(* IEC 61131-3 sources: beckhoffAutomationInterface/ST/Shark/Lib/Sequences/SubSequence, 11 files *)

(* ---- FB_BubblerPurgeCMSequence.st ---- *)
FUNCTION_BLOCK PUBLIC FB_BubblerPurgeCMSequence IMPLEMENTS I_TreeNode
VAR
    _seq : FB_SequenceNode;
    // Steps
    stepOpenBubbler  : FB_OpenValveNode;
    stepPurgeCM      : FB_MaterialPurgeCMSequence;
    stepCloseBubbler : FB_CloseValveNode;

    // Internal state
    _bInitialized    : BOOL := FALSE;
    _eSide           : E_GasSide;
    _nBubblerIndex   : DINT;
END_VAR

METHOD PUBLIC Init : BOOL
VAR_INPUT
    ipProvider      : I_HardwareProvider;
    eSide           : E_GasSide;
    nBubblerIndex   : DINT;
END_VAR
VAR
    ipCMBubblerValve : I_Valve;
END_VAR
    IF _bInitialized THEN
        IF _eSide = eSide AND _nBubblerIndex = nBubblerIndex THEN
            Init := TRUE;
            RETURN;
        END_IF
        _seq.ClearChildren();
        _bInitialized := FALSE;
    END_IF

    IF ipProvider = 0 THEN
        GVL_ErrorLogger.Logger.LogError('FB_BubblerPurgeCMSequence', E_ErrorId.ERR_GEN_NULL_POINTER, 'Provider is null');
        RETURN;
    END_IF
    _eSide := eSide;
    _nBubblerIndex := nBubblerIndex;

    // Resolve hardware
    ipCMBubblerValve := ipProvider.GetCMBubblerValve(eSide, nBubblerIndex);

    IF ipCMBubblerValve = 0 THEN
        GVL_ErrorLogger.Logger.LogError('FB_BubblerPurgeCMSequence', E_ErrorId.ERR_GEN_NULL_POINTER, 'Bubbler Valve not found');
        RETURN;
    END_IF

    stepOpenBubbler.Init(ipCMBubblerValve, sNodeName := 'OpenBubblerCMValve');
    _seq.AddChild(stepOpenBubbler);

    stepPurgeCM.Init(ipProvider, eSide);
    stepPurgeCM.NodeName := 'PurgeCMSequence';
    _seq.AddChild(stepPurgeCM);

    stepCloseBubbler.Init(ipCMBubblerValve, sNodeName := 'CloseBubblerCMValve');
    _seq.AddChild(stepCloseBubbler);

    _seq.sName := CONCAT('BubblerPurgeCM_Side', TO_STRING(eSide));
    _bInitialized := TRUE;
    Init := TRUE;
END_METHOD

METHOD PUBLIC SetParams
VAR_INPUT
    nPurgeCycles            : INT;
    rPurgeFlowRate          : LREAL;
    rPurgePressure          : LREAL;
    rEvacuationPressure     : LREAL;
    tPressurizationTimeout  : TIME;
    tEvacuationTimeout      : TIME;
END_VAR
    IF NOT _bInitialized THEN RETURN; END_IF

    stepPurgeCM.SetParams(
        nPurgeCycles           := nPurgeCycles,
        rPurgeFlowRate         := rPurgeFlowRate,
        rPurgePressure         := rPurgePressure,
        rEvacuationPressure    := rEvacuationPressure,
        tPressurizationTimeout := tPressurizationTimeout,
        tEvacuationTimeout     := tEvacuationTimeout
    );
END_METHOD

PROPERTY PUBLIC NodeName : STRING(50)
    GET
        NodeName := _seq.sName;
    END_GET
    SET
        _seq.sName := NodeName;
    END_SET
END_PROPERTY

METHOD Tick : ST_NodeResult
    IF NOT _bInitialized THEN
        Tick.eStatus := E_NodeStatus.FAILURE;
        Tick.bHasError := TRUE;
        Tick.stError.eErrorId := E_ErrorId.ERR_GEN_INITIALIZATION;
        Tick.stError.sSource := 'FB_BubblerPurgeCMSequence';
        Tick.stError.sMessage := 'Init must be called before Tick';
        Tick.sDescription := Tick.stError.sMessage;
        RETURN;
    END_IF

    Tick := _seq.Tick();
END_METHOD

{attribute 'estimated-stack-usage' := '500'}
METHOD Reset : BOOL
    Reset := _seq.Reset();
END_METHOD

{attribute 'estimated-stack-usage' := '500'}
METHOD Halt
    _seq.Halt();
END_METHOD

END_FUNCTION_BLOCK

(* ---- FB_BubblerPurgeHMSequence.st ---- *)
FUNCTION_BLOCK PUBLIC FB_BubblerPurgeHMSequence IMPLEMENTS I_TreeNode
VAR
    _seq : FB_SequenceNode;
    // Steps
    stepOpenBubbler  : FB_OpenValveNode;
    stepPurgeHM      : FB_MaterialPurgeHMSequence;
    stepCloseBubbler : FB_CloseValveNode;

    // Internal state
    _bInitialized    : BOOL := FALSE;
    _eSide           : E_GasSide;
    _nBubblerIndex   : DINT;
END_VAR

METHOD PUBLIC Init : BOOL
VAR_INPUT
    ipProvider      : I_HardwareProvider;
    eSide           : E_GasSide;
    nBubblerIndex   : DINT;
END_VAR
VAR
    ipHMBubblerValve : I_Valve;
END_VAR
    IF _bInitialized THEN
        IF _eSide = eSide AND _nBubblerIndex = nBubblerIndex THEN
            Init := TRUE;
            RETURN;
        END_IF
        _seq.ClearChildren();
        _bInitialized := FALSE;
    END_IF

    IF ipProvider = 0 THEN
        GVL_ErrorLogger.Logger.LogError('FB_BubblerPurgeHMSequence', E_ErrorId.ERR_GEN_NULL_POINTER, 'Provider is null');
        RETURN;
    END_IF
    _eSide := eSide;
    _nBubblerIndex := nBubblerIndex;

    // Resolve hardware
    ipHMBubblerValve := ipProvider.GetHMBubblerValve(eSide, nBubblerIndex);

    IF ipHMBubblerValve = 0 THEN
        GVL_ErrorLogger.Logger.LogError('FB_BubblerPurgeHMSequence', E_ErrorId.ERR_GEN_NULL_POINTER, 'Bubbler Valve not found');
        RETURN;
    END_IF

    stepOpenBubbler.Init(ipHMBubblerValve, sNodeName := 'OpenBubblerHMValve');
    _seq.AddChild(stepOpenBubbler);

    stepPurgeHM.Init(ipProvider, eSide);
    stepPurgeHM.NodeName := 'PurgeHMSequence';
    _seq.AddChild(stepPurgeHM);

    stepCloseBubbler.Init(ipHMBubblerValve, sNodeName := 'CloseBubblerHMValve');
    _seq.AddChild(stepCloseBubbler);

    _seq.sName := CONCAT('BubblerPurgeHM_Side', TO_STRING(eSide));
    _bInitialized := TRUE;
    Init := TRUE;
END_METHOD

METHOD PUBLIC SetParams
VAR_INPUT
    nPurgeCycles            : INT;
    rPurgeFlowRate          : LREAL;
    rPurgePressure          : LREAL;
    rFinalPressure          : LREAL;   // Operating pressure for final pressurization
    rEvacuationPressure     : LREAL;
    tPressurizationTimeout  : TIME;
    tEvacuationTimeout      : TIME;
END_VAR
    IF NOT _bInitialized THEN RETURN; END_IF

    stepPurgeHM.SetParams(
        nPurgeCycles           := nPurgeCycles,
        rPurgeFlowRate         := rPurgeFlowRate,
        rPurgePressure         := rPurgePressure,
        rFinalPressure         := rFinalPressure,
        rEvacuationPressure    := rEvacuationPressure,
        tPressurizationTimeout := tPressurizationTimeout,
        tEvacuationTimeout     := tEvacuationTimeout
    );
END_METHOD

PROPERTY PUBLIC NodeName : STRING(50)
    GET
        NodeName := _seq.sName;
    END_GET
    SET
        _seq.sName := NodeName;
    END_SET
END_PROPERTY

METHOD Tick : ST_NodeResult
    IF NOT _bInitialized THEN
        Tick.eStatus := E_NodeStatus.FAILURE;
        Tick.bHasError := TRUE;
        Tick.stError.eErrorId := E_ErrorId.ERR_GEN_INITIALIZATION;
        Tick.stError.sSource := 'FB_BubblerPurgeHMSequence';
        Tick.stError.sMessage := 'Init must be called before Tick';
        Tick.sDescription := Tick.stError.sMessage;
        RETURN;
    END_IF

    Tick := _seq.Tick();
END_METHOD

{attribute 'estimated-stack-usage' := '500'}
METHOD Reset : BOOL
    Reset := _seq.Reset();
END_METHOD

{attribute 'estimated-stack-usage' := '500'}
METHOD Halt
    _seq.Halt();
END_METHOD

END_FUNCTION_BLOCK

(* ---- FB_DepressurizeCMSequence.st ---- *)
FUNCTION_BLOCK PUBLIC FB_DepressurizeCMSequence IMPLEMENTS I_TreeNode
VAR
    _seq : FB_SequenceNode;
    // Steps
    stepOpenCMPurge      : FB_OpenValveNode;
    stepOpenCMVacuumIso  : FB_OpenValveNode;
    stepWaitCMVacuum     : FB_WaitForSensorNode;
    stepCloseCMVacuumIso : FB_CloseValveNode;
    stepCloseCMPurge     : FB_CloseValveNode;

    // Internal state
    _bInitialized        : BOOL := FALSE;
    _eSide               : E_GasSide;
END_VAR

VAR CONSTANT
    DEFAULT_VACUUM_THRESHOLD : LREAL := 1.0; // Bar - pressure below which vacuum is considered achieved
END_VAR

METHOD PUBLIC Init : BOOL
VAR_INPUT
    ipProvider     : I_HardwareProvider;
    eSide          : E_GasSide;
    tVacuumTimeout : TIME := T#30S;
END_VAR
VAR
    ipCMPurge     : I_Valve;
    ipCMVacuumIso : I_Valve;
    ipCMPressure  : I_Sensor;
END_VAR
    IF _bInitialized THEN
        IF _eSide = eSide THEN
            Init := TRUE;
            RETURN;
        END_IF
        _seq.ClearChildren();
        _bInitialized := FALSE;
    END_IF

    IF ipProvider = 0 THEN
        GVL_ErrorLogger.Logger.LogError('FB_DepressurizeCMSequence', E_ErrorId.ERR_GEN_NULL_POINTER, 'Provider is null');
        RETURN;
    END_IF
    _eSide := eSide;

    // Resolve hardware references
    ipCMPurge := ipProvider.GetCMPurgeValve(eSide);
    ipCMVacuumIso := ipProvider.GetCMVacuumIsoValve(eSide);
    ipCMPressure := ipProvider.GetCMPressureSensor(eSide);

    IF ipCMPurge = 0 OR ipCMVacuumIso = 0 OR ipCMPressure = 0 THEN
        GVL_ErrorLogger.Logger.LogError('FB_DepressurizeCMSequence', E_ErrorId.ERR_GEN_NULL_POINTER, 'Hardware reference is null');
        RETURN;
    END_IF

    // Evacuation: open path to exhaust, wait for vacuum, then close
    stepOpenCMPurge.Init(ipCMPurge, sNodeName := 'OpenCMPurge');
    _seq.AddChild(stepOpenCMPurge);

    stepOpenCMVacuumIso.Init(ipCMVacuumIso, sNodeName := 'OpenCMVacuumIso');
    _seq.AddChild(stepOpenCMVacuumIso);

    stepWaitCMVacuum.Init(
        ipSensor    := ipCMPressure,
        rTarget     := DEFAULT_VACUUM_THRESHOLD,
        eMode       := E_CompareMode.LESS_THAN,
        tTimeout    := tVacuumTimeout,
        sNodeName   := 'WaitCMVacuum'
    );
    _seq.AddChild(stepWaitCMVacuum);

    stepCloseCMVacuumIso.Init(ipCMVacuumIso, sNodeName := 'CloseCMVacuumIso');
    _seq.AddChild(stepCloseCMVacuumIso);

    stepCloseCMPurge.Init(ipCMPurge, sNodeName := 'CloseCMPurge');
    _seq.AddChild(stepCloseCMPurge);

    _seq.sName := CONCAT('DepressurizeCM_', TO_STRING(eSide));
    _bInitialized := TRUE;
    Init := TRUE;
END_METHOD

METHOD PUBLIC SetParams
VAR_INPUT
    rVacuumThreshold : LREAL;
    tTimeout         : TIME;
END_VAR
    IF NOT _bInitialized THEN RETURN; END_IF

    stepWaitCMVacuum.Target := rVacuumThreshold;
    stepWaitCMVacuum.Timeout := tTimeout;
END_METHOD

PROPERTY PUBLIC NodeName : STRING(50)
    GET
        NodeName := _seq.sName;
    END_GET
    SET
        _seq.sName := NodeName;
    END_SET
END_PROPERTY

METHOD Tick : ST_NodeResult
    IF NOT _bInitialized THEN
        Tick.eStatus := E_NodeStatus.FAILURE;
        Tick.bHasError := TRUE;
        Tick.stError.eErrorId := E_ErrorId.ERR_GEN_INITIALIZATION;
        Tick.stError.sSource := 'FB_DepressurizeCMSequence';
        Tick.stError.sMessage := 'Init must be called before Tick';
        Tick.sDescription := Tick.stError.sMessage;
        RETURN;
    END_IF

    Tick := _seq.Tick();
END_METHOD

{attribute 'estimated-stack-usage' := '500'}
METHOD Reset : BOOL
    Reset := _seq.Reset();
END_METHOD

{attribute 'estimated-stack-usage' := '500'}
METHOD Halt
    _seq.Halt();
END_METHOD

END_FUNCTION_BLOCK

(* ---- FB_DepressurizeHMSequence.st ---- *)
FUNCTION_BLOCK PUBLIC FB_DepressurizeHMSequence IMPLEMENTS I_TreeNode
VAR
    _seq : FB_SequenceNode;
    // Safety steps
    stepCloseNozzle      : FB_CloseValveNode;
    stepClosePCV         : FB_SetControllerNode;

    // Evacuation
    stepOpenHMVacuumIso  : FB_OpenValveNode;
    stepOpenHMPurge      : FB_OpenValveNode;
    stepWaitHMVacuum     : FB_WaitForSensorNode;
    stepCloseHMVacuumIso : FB_CloseValveNode;
    stepCloseHMPurge     : FB_CloseValveNode;

    // Internal state
    _bInitialized        : BOOL := FALSE;
    _eSide               : E_GasSide;
END_VAR

VAR CONSTANT
    DEFAULT_VACUUM_THRESHOLD : LREAL := 1.0; // Bar - pressure below which vacuum is considered achieved
END_VAR

METHOD PUBLIC Init : BOOL
VAR_INPUT
    ipProvider    : I_HardwareProvider;
    eSide         : E_GasSide;
    tVacuumTimeout : TIME := T#30S;
END_VAR
VAR
    ipNozzleIso   : I_Valve;
    ipPCV         : I_Controller;
    ipHMPurge     : I_Valve;
    ipHMVacuumIso : I_Valve;
    ipHMPressure  : I_Sensor;
END_VAR
    IF _bInitialized THEN
        IF _eSide = eSide THEN
            Init := TRUE;
            RETURN;
        END_IF
        _seq.ClearChildren();
        _bInitialized := FALSE;
    END_IF

    IF ipProvider = 0 THEN
        GVL_ErrorLogger.Logger.LogError('FB_DepressurizeHMSequence', E_ErrorId.ERR_GEN_NULL_POINTER, 'Provider is null');
        RETURN;
    END_IF
    _eSide := eSide;

    // Resolve hardware references
    ipNozzleIso := ipProvider.GetNozzleIsoValve(eSide);
    ipPCV := ipProvider.GetPressureController(eSide);
    ipHMPurge := ipProvider.GetHMPurgeValve(eSide);
    ipHMVacuumIso := ipProvider.GetHMVacuumIsoValve(eSide);
    ipHMPressure := ipProvider.GetHMPressureSensor(eSide);

    IF ipNozzleIso = 0 OR ipPCV = 0 OR ipHMPurge = 0 OR ipHMVacuumIso = 0 OR ipHMPressure = 0 THEN
        GVL_ErrorLogger.Logger.LogError('FB_DepressurizeHMSequence', E_ErrorId.ERR_GEN_NULL_POINTER, 'Hardware reference is null');
        RETURN;
    END_IF

    // Safety: isolate nozzle and close PCV
    stepCloseNozzle.Init(ipNozzleIso, sNodeName := 'CloseNozzle');
    _seq.AddChild(stepCloseNozzle);

    stepClosePCV.Init(ipController := ipPCV, rSetpoint := GVL_SequenceConstants.PCV_CLOSED_SETPOINT, sNodeName := 'ClosePCV');
    _seq.AddChild(stepClosePCV);

    // Evacuation: open path to exhaust, wait for vacuum, then close
    stepOpenHMVacuumIso.Init(ipHMVacuumIso, sNodeName := 'OpenHMVacuumIso');
    _seq.AddChild(stepOpenHMVacuumIso);

    stepOpenHMPurge.Init(ipHMPurge, sNodeName := 'OpenHMPurge');
    _seq.AddChild(stepOpenHMPurge);

    stepWaitHMVacuum.Init(
        ipSensor    := ipHMPressure,
        rTarget     := DEFAULT_VACUUM_THRESHOLD,
        eMode       := E_CompareMode.LESS_THAN,
        tTimeout    := tVacuumTimeout,
        sNodeName   := 'WaitHMVacuum'
    );
    _seq.AddChild(stepWaitHMVacuum);

    stepCloseHMPurge.Init(ipHMPurge, sNodeName := 'CloseHMPurge');
    _seq.AddChild(stepCloseHMPurge);

    stepCloseHMVacuumIso.Init(ipHMVacuumIso, sNodeName := 'CloseHMVacuumIso');
    _seq.AddChild(stepCloseHMVacuumIso);

    _seq.sName := CONCAT('DepressurizeHM_', TO_STRING(eSide));
    _bInitialized := TRUE;
    Init := TRUE;
END_METHOD

METHOD PUBLIC SetParams
VAR_INPUT
    rVacuumThreshold : LREAL;
    tTimeout         : TIME;
END_VAR
    IF NOT _bInitialized THEN RETURN; END_IF

    stepWaitHMVacuum.Target := rVacuumThreshold;
    stepWaitHMVacuum.Timeout := tTimeout;
END_METHOD

PROPERTY PUBLIC NodeName : STRING(50)
    GET
        NodeName := _seq.sName;
    END_GET
    SET
        _seq.sName := NodeName;
    END_SET
END_PROPERTY

METHOD Tick : ST_NodeResult
    IF NOT _bInitialized THEN
        Tick.eStatus := E_NodeStatus.FAILURE;
        Tick.bHasError := TRUE;
        Tick.stError.eErrorId := E_ErrorId.ERR_GEN_INITIALIZATION;
        Tick.stError.sSource := 'FB_DepressurizeHMSequence';
        Tick.stError.sMessage := 'Init must be called before Tick';
        Tick.sDescription := Tick.stError.sMessage;
        RETURN;
    END_IF

    Tick := _seq.Tick();
END_METHOD

{attribute 'estimated-stack-usage' := '500'}
METHOD Reset : BOOL
    Reset := _seq.Reset();
END_METHOD

{attribute 'estimated-stack-usage' := '500'}
METHOD Halt
    _seq.Halt();
END_METHOD

END_FUNCTION_BLOCK

(* ---- FB_MaintenancePurgeUmbilicalSequence.st ---- *)
(*
FB_MaintenancePurgeUmbilicalSequence
Purges the umbilical region (PCV->Nozzle) by pushing inert gas to atmosphere.
Flow path: Gas->MFC->CM Purge->HM Purge->HM->PCV->Nozzle->Atmosphere
Pressure builds CM->HM sequentially to prevent reactive gas backflow.
*)
FUNCTION_BLOCK PUBLIC FB_MaintenancePurgeUmbilicalSequence IMPLEMENTS I_TreeNode
VAR
    _seq : FB_SequenceNode;
    // Phase 1: Preparation
    stepCloseNozzleIso     : FB_CloseValveNode;
    stepClosePCV           : FB_SetControllerNode;

    // Phase 2: Pressurize via purge bypass (CM->HM to prevent backflow)
    stepOpenGasIso         : FB_OpenValveNode;
    stepSetMFC             : FB_SetControllerNode;
    stepOpenCMPurge        : FB_OpenValveNode;
    stepWaitForCMPressure  : FB_WaitForSensorNode;
    stepOpenHMPurge        : FB_OpenValveNode;
    stepWaitForHMPressure  : FB_WaitForSensorNode;

    // Phase 3: Purge to atmosphere
    stepSetPCV             : FB_SetControllerNode;
    stepStabilizationDelay : FB_WaitNode;
    stepOpenNozzleIso      : FB_OpenValveNode;
    stepPurgeDuration      : FB_WaitNode;

    // Phase 4: Cleanup
    stepCleanup            : FB_SequenceNode;
    stepCloseNozzleIsoFinal: FB_CloseValveNode;
    stepClosePCVFinal      : FB_SetControllerNode;
    stepStopMFC            : FB_SetControllerNode;
    stepCloseGasIso        : FB_CloseValveNode;
    stepCloseCMPurge       : FB_CloseValveNode;
    stepCloseHMPurge       : FB_CloseValveNode;

    // Internal state
    _bInitialized          : BOOL := FALSE;
    _bParamsConfigured     : BOOL := FALSE;
    _eSide                 : E_GasSide;
END_VAR

VAR CONSTANT
    DEFAULT_STABILIZATION_DELAY : TIME := T#5S;
    DEFAULT_PURGE_DURATION      : TIME := T#30S;
END_VAR

METHOD PUBLIC Init : BOOL
VAR_INPUT
    ipProvider : I_HardwareProvider;
    eSide      : E_GasSide;
END_VAR
VAR
    ipGasIso      : I_Valve;
    ipMFC         : I_Controller;
    ipCMPurge     : I_Valve;
    ipCMPressure  : I_Sensor;
    ipHMPurge     : I_Valve;
    ipHMPressure  : I_Sensor;
    ipPCV         : I_Controller;
    ipNozzleIso   : I_Valve;
END_VAR
    IF _bInitialized THEN
        IF _eSide = eSide THEN
            Init := TRUE;
            RETURN;
        END_IF
        _seq.ClearChildren();
        stepCleanup.ClearChildren();
        _bInitialized := FALSE;
    END_IF

    IF ipProvider = 0 THEN
        GVL_ErrorLogger.Logger.LogError('FB_MaintenancePurgeUmbilicalSequence', E_ErrorId.ERR_GEN_NULL_POINTER, 'Provider is null');
        RETURN;
    END_IF
    _eSide := eSide;

    // Resolve hardware
    ipGasIso := ipProvider.GetGasIsoValve(eSide, 0);
    ipMFC := ipProvider.GetMFCController(eSide);
    ipCMPurge := ipProvider.GetCMPurgeValve(eSide);
    ipCMPressure := ipProvider.GetCMPressureSensor(eSide);
    ipHMPurge := ipProvider.GetHMPurgeValve(eSide);
    ipHMPressure := ipProvider.GetHMPressureSensor(eSide);
    ipPCV := ipProvider.GetPressureController(eSide);
    ipNozzleIso := ipProvider.GetNozzleIsoValve(eSide);

    // Validate hardware
    IF ipGasIso = 0 OR ipMFC = 0 OR ipCMPurge = 0 OR ipCMPressure = 0 OR
       ipHMPurge = 0 OR ipHMPressure = 0 OR ipPCV = 0 OR ipNozzleIso = 0 THEN
        GVL_ErrorLogger.Logger.LogError('FB_MaintenancePurgeUmbilicalSequence', E_ErrorId.ERR_GEN_NULL_POINTER, 'Hardware reference is null');
        RETURN;
    END_IF

    // Phase 1: Preparation
    stepCloseNozzleIso.Init(ipNozzleIso, sNodeName := 'CloseNozzleIso');
    _seq.AddChild(stepCloseNozzleIso);

    stepClosePCV.Init(ipController := ipPCV, rSetpoint := GVL_SequenceConstants.PCV_CLOSED_SETPOINT, sNodeName := 'ClosePCV');
    _seq.AddChild(stepClosePCV);

    // Phase 2: Pressurize via purge bypass (CM->HM to prevent backflow)
    stepOpenGasIso.Init(ipGasIso, sNodeName := 'OpenGasIso');
    _seq.AddChild(stepOpenGasIso);

    stepSetMFC.Init(ipController := ipMFC, rSetpoint := 0.0, sNodeName := 'SetPurgeMFC');
    _seq.AddChild(stepSetMFC);

    stepOpenCMPurge.Init(ipCMPurge, sNodeName := 'OpenCMPurge');
    _seq.AddChild(stepOpenCMPurge);

    stepWaitForCMPressure.Init(ipSensor := ipCMPressure, rTarget := 0.0, eMode := E_CompareMode.GREATER_THAN, sNodeName := 'WaitForCMPressure');
    _seq.AddChild(stepWaitForCMPressure);

    stepOpenHMPurge.Init(ipHMPurge, sNodeName := 'OpenHMPurge');
    _seq.AddChild(stepOpenHMPurge);

    stepWaitForHMPressure.Init(ipSensor := ipHMPressure, rTarget := 0.0, eMode := E_CompareMode.GREATER_THAN, sNodeName := 'WaitForHMPressure');
    _seq.AddChild(stepWaitForHMPressure);

    // Phase 3: Purge to atmosphere
    stepSetPCV.Init(ipController := ipPCV, rSetpoint := 0.0, sNodeName := 'SetPCVSetpoint');
    _seq.AddChild(stepSetPCV);

    stepStabilizationDelay.Init(tWaitTime := DEFAULT_STABILIZATION_DELAY, sNodeName := 'StabilizationDelay');
    _seq.AddChild(stepStabilizationDelay);

    stepOpenNozzleIso.Init(ipNozzleIso, sNodeName := 'OpenNozzleIso');
    _seq.AddChild(stepOpenNozzleIso);

    stepPurgeDuration.Init(tWaitTime := DEFAULT_PURGE_DURATION, sNodeName := 'PurgeDuration');
    _seq.AddChild(stepPurgeDuration);

    // Phase 4: Cleanup
    stepCleanup.ClearChildren();

    stepCloseNozzleIsoFinal.Init(ipNozzleIso, sNodeName := 'CloseNozzleIsoFinal');
    stepCleanup.AddChild(stepCloseNozzleIsoFinal);

    stepClosePCVFinal.Init(ipController := ipPCV, rSetpoint := GVL_SequenceConstants.PCV_CLOSED_SETPOINT, sNodeName := 'ClosePCVFinal');
    stepCleanup.AddChild(stepClosePCVFinal);

    stepStopMFC.Init(ipController := ipMFC, rSetpoint := 0.0, sNodeName := 'StopMFC');
    stepCleanup.AddChild(stepStopMFC);

    stepCloseGasIso.Init(ipGasIso, sNodeName := 'CloseGasIso');
    stepCleanup.AddChild(stepCloseGasIso);

    stepCloseCMPurge.Init(ipCMPurge, sNodeName := 'CloseCMPurge');
    stepCleanup.AddChild(stepCloseCMPurge);

    stepCloseHMPurge.Init(ipHMPurge, sNodeName := 'CloseHMPurge');
    stepCleanup.AddChild(stepCloseHMPurge);

    stepCleanup.sName := 'Cleanup';
    _seq.AddChild(stepCleanup);

    _seq.sName := CONCAT('MaintUmbilicalPurge_', TO_STRING(eSide));
    _bParamsConfigured := FALSE;
    _bInitialized := TRUE;
    Init := TRUE;
END_METHOD

METHOD PUBLIC SetParams
VAR_INPUT
    rPurgeFlowRate      : LREAL;    // MFC flow rate during purge (sccm/slm)
    rCMPressureTarget   : LREAL;    // CM pressure target before opening HM Purge (bar)
    rHMPressureTarget   : LREAL;    // HM pressure target before opening nozzle (bar)
    rPCVSetpoint        : LREAL;    // PCV setpoint during purge (bar)
    tCMPressureTimeout  : TIME;     // Timeout for CM pressure build
    tHMPressureTimeout  : TIME;     // Timeout for HM pressure build
    tStabilizationDelay : TIME;     // Delay after setting PCV
    tPurgeDuration      : TIME;     // Duration of purge to atmosphere
END_VAR
    IF NOT _bInitialized THEN RETURN; END_IF

    stepSetMFC.Setpoint := rPurgeFlowRate;

    stepWaitForCMPressure.Target := rCMPressureTarget;
    stepWaitForCMPressure.Timeout := tCMPressureTimeout;

    stepWaitForHMPressure.Target := rHMPressureTarget;
    stepWaitForHMPressure.Timeout := tHMPressureTimeout;

    stepSetPCV.Setpoint := rPCVSetpoint;

    stepStabilizationDelay.WaitTime := tStabilizationDelay;
    stepPurgeDuration.WaitTime := tPurgeDuration;
    _bParamsConfigured := TRUE;
END_METHOD

PROPERTY PUBLIC NodeName : STRING(50)
    GET
        NodeName := _seq.sName;
    END_GET
    SET
        _seq.sName := NodeName;
    END_SET
END_PROPERTY

METHOD Tick : ST_NodeResult
    IF NOT _bInitialized THEN
        Tick.eStatus := E_NodeStatus.FAILURE;
        Tick.bHasError := TRUE;
        Tick.stError.eErrorId := E_ErrorId.ERR_GEN_INITIALIZATION;
        Tick.stError.sSource := 'FB_MaintenancePurgeUmbilicalSequence';
        Tick.stError.sMessage := 'Init must be called before Tick';
        Tick.sDescription := Tick.stError.sMessage;
        RETURN;
    END_IF

    IF NOT _bParamsConfigured THEN
        Tick.eStatus := E_NodeStatus.FAILURE;
        Tick.bHasError := TRUE;
        Tick.stError.eErrorId := E_ErrorId.ERR_GEN_NOT_CONFIGURED;
        Tick.stError.sSource := 'FB_MaintenancePurgeUmbilicalSequence';
        Tick.stError.sMessage := 'SetParams must be called before Tick';
        Tick.sDescription := Tick.stError.sMessage;
        RETURN;
    END_IF

    Tick := _seq.Tick();
END_METHOD

{attribute 'estimated-stack-usage' := '500'}
METHOD Reset : BOOL
    Reset := _seq.Reset();
END_METHOD

{attribute 'estimated-stack-usage' := '500'}
METHOD Halt
    _seq.Halt();
END_METHOD

END_FUNCTION_BLOCK

(* ---- FB_MaterialPurgeCMSequence.st ---- *)
FUNCTION_BLOCK PUBLIC FB_MaterialPurgeCMSequence IMPLEMENTS I_TreeNode
VAR
    _seq : FB_SequenceNode;
    // Purge cycle structure
    stepPurgeCycles        : FB_RepeatNode;
    stepPurgeCycleSeq      : FB_SequenceNode;

    // Fill steps
    stepOpenExhaustVacIso  : FB_OpenValveNode;
    stepOpenGasIso         : FB_OpenValveNode;
    stepSetMFC             : FB_SetControllerNode;
    stepOpenCMPurge        : FB_OpenValveNode;
    stepCloseCMPurge       : FB_CloseValveNode;
    stepWaitForFill        : FB_WaitForSensorNode;

    // Dump steps
    stepStopFillMFC        : FB_SetControllerNode;
    stepCloseGasIsoForDump : FB_CloseValveNode;
    stepOpenCMVacuumIso    : FB_OpenValveNode;
    stepCloseCMVacuumIso   : FB_CloseValveNode;
    stepWaitForDump        : FB_WaitForSensorNode;

    // Cleanup
    stepCloseGasIsoFinal      : FB_CloseValveNode;
    stepCloseCMPurgeFinal     : FB_CloseValveNode;
    stepCloseCMVacuumIsoFinal : FB_CloseValveNode;

    // Internal state
    _bInitialized          : BOOL := FALSE;
    _bParamsConfigured     : BOOL := FALSE;
    _eSide                 : E_GasSide;
END_VAR

VAR CONSTANT
    DEFAULT_PURGE_CYCLES   : INT := 3;
    DEFAULT_DUMP_THRESHOLD : LREAL := 1.0; // Bar - pressure below which dump is considered complete
END_VAR

METHOD PUBLIC Init : BOOL
VAR_INPUT
    ipProvider      : I_HardwareProvider;
    eSide           : E_GasSide;
END_VAR
VAR
    ipGasIso         : I_Valve;
    ipCMPurge        : I_Valve;
    ipCMPressure     : I_Sensor;
    ipCMVacuumIso    : I_Valve;
    ipMFC            : I_Controller;
END_VAR
    IF _bInitialized THEN
        IF _eSide = eSide THEN
            Init := TRUE;
            RETURN;
        END_IF
        _seq.ClearChildren();
        stepPurgeCycleSeq.ClearChildren();
        _bInitialized := FALSE;
    END_IF

    IF ipProvider = 0 THEN
        GVL_ErrorLogger.Logger.LogError('FB_MaterialPurgeCMSequence', E_ErrorId.ERR_GEN_NULL_POINTER, 'Provider is null');
        RETURN;
    END_IF
    _eSide := eSide;

    // Resolve hardware
    ipMFC := ipProvider.GetMFCController(eSide);
    ipGasIso := ipProvider.GetGasIsoValve(eSide, 0);
    ipCMPurge := ipProvider.GetCMPurgeValve(eSide);
    ipCMPressure := ipProvider.GetCMPressureSensor(eSide);
    ipCMVacuumIso := ipProvider.GetCMVacuumIsoValve(eSide);

    // Validate hardware
    IF ipMFC = 0 OR ipGasIso = 0 OR ipCMPurge = 0 OR ipCMPressure = 0 OR ipCMVacuumIso = 0 THEN
        GVL_ErrorLogger.Logger.LogError('FB_MaterialPurgeCMSequence', E_ErrorId.ERR_GEN_NULL_POINTER, 'Hardware reference is null');
        RETURN;
    END_IF

    // Precondition: ensure exhaust path is open
    stepOpenExhaustVacIso.Init(ipProvider.GetExhaustVacuumIsoValve(), sNodeName := 'OpenExhaustVacIso');
    _seq.AddChild(stepOpenExhaustVacIso);

    // Build purge cycle: fill then dump
    stepCloseCMVacuumIso.Init(ipCMVacuumIso, sNodeName := 'EnsureCMVacuumIsoClosed');
    stepPurgeCycleSeq.AddChild(stepCloseCMVacuumIso);

    stepOpenGasIso.Init(ipGasIso, sNodeName := 'OpenGasIso');
    stepPurgeCycleSeq.AddChild(stepOpenGasIso);

    stepSetMFC.Init(ipController := ipMFC, rSetpoint := 0.0, sNodeName := 'SetPurgeMFC');
    stepPurgeCycleSeq.AddChild(stepSetMFC);

    stepOpenCMPurge.Init(ipCMPurge, sNodeName := 'OpenCMPurge');
    stepPurgeCycleSeq.AddChild(stepOpenCMPurge);

    stepWaitForFill.Init(ipSensor := ipCMPressure, rTarget := 0.0, eMode := E_CompareMode.GREATER_THAN, sNodeName := 'WaitForCMFill');
    stepPurgeCycleSeq.AddChild(stepWaitForFill);

    stepStopFillMFC.Init(ipController := ipMFC, rSetpoint := 0.0, sNodeName := 'StopMFC');
    stepPurgeCycleSeq.AddChild(stepStopFillMFC);

    stepCloseGasIsoForDump.Init(ipGasIso, sNodeName := 'CloseGasIso');
    stepPurgeCycleSeq.AddChild(stepCloseGasIsoForDump);

    stepOpenCMVacuumIso.Init(ipCMVacuumIso, sNodeName := 'OpenCMVacuumIso');
    stepPurgeCycleSeq.AddChild(stepOpenCMVacuumIso);

    stepWaitForDump.Init(ipSensor := ipCMPressure, rTarget := DEFAULT_DUMP_THRESHOLD, eMode := E_CompareMode.LESS_THAN, sNodeName := 'WaitForCMDump');
    stepPurgeCycleSeq.AddChild(stepWaitForDump);

    stepPurgeCycles.SetChild(stepPurgeCycleSeq);
    stepPurgeCycles.nNumCycles := DEFAULT_PURGE_CYCLES;
    stepPurgeCycles.sName := 'CMPurgeCycles';
    _seq.AddChild(stepPurgeCycles);

    // Cleanup
    stepCloseGasIsoFinal.Init(ipGasIso, sNodeName := 'CloseGasIsoFinal');
    _seq.AddChild(stepCloseGasIsoFinal);

    stepCloseCMPurgeFinal.Init(ipCMPurge, sNodeName := 'CloseCMPurgeFinal');
    _seq.AddChild(stepCloseCMPurgeFinal);

    stepCloseCMVacuumIsoFinal.Init(ipCMVacuumIso, sNodeName := 'CloseCMVacuumIsoFinal');
    _seq.AddChild(stepCloseCMVacuumIsoFinal);

    _seq.sName := CONCAT('PurgeCM_', TO_STRING(eSide));
    _bParamsConfigured := FALSE;
    _bInitialized := TRUE;
    Init := TRUE;
END_METHOD

METHOD PUBLIC SetParams
VAR_INPUT
    nPurgeCycles            : INT;
    rPurgeFlowRate          : LREAL;
    rPurgePressure          : LREAL;
    rEvacuationPressure     : LREAL;
    tPressurizationTimeout  : TIME;
    tEvacuationTimeout      : TIME;
END_VAR
    IF NOT _bInitialized THEN RETURN; END_IF

    stepPurgeCycles.nNumCycles := nPurgeCycles;
    stepSetMFC.Setpoint := rPurgeFlowRate;
    stepWaitForFill.Target := rPurgePressure;
    stepWaitForFill.Timeout := tPressurizationTimeout;
    stepWaitForDump.Target := rEvacuationPressure;
    stepWaitForDump.Timeout := tEvacuationTimeout;
    _bParamsConfigured := TRUE;
END_METHOD

PROPERTY PUBLIC NodeName : STRING(50)
    GET
        NodeName := _seq.sName;
    END_GET
    SET
        _seq.sName := NodeName;
    END_SET
END_PROPERTY

METHOD Tick : ST_NodeResult
    IF NOT _bInitialized THEN
        Tick.eStatus := E_NodeStatus.FAILURE;
        Tick.bHasError := TRUE;
        Tick.stError.eErrorId := E_ErrorId.ERR_GEN_INITIALIZATION;
        Tick.stError.sSource := 'FB_MaterialPurgeCMSequence';
        Tick.stError.sMessage := 'Init must be called before Tick';
        Tick.sDescription := Tick.stError.sMessage;
        RETURN;
    END_IF

    IF NOT _bParamsConfigured THEN
        Tick.eStatus := E_NodeStatus.FAILURE;
        Tick.bHasError := TRUE;
        Tick.stError.eErrorId := E_ErrorId.ERR_GEN_NOT_CONFIGURED;
        Tick.stError.sSource := 'FB_MaterialPurgeCMSequence';
        Tick.stError.sMessage := 'SetParams must be called before Tick';
        Tick.sDescription := Tick.stError.sMessage;
        RETURN;
    END_IF

    Tick := _seq.Tick();
END_METHOD

{attribute 'estimated-stack-usage' := '500'}
METHOD Reset : BOOL
    Reset := _seq.Reset();
END_METHOD

{attribute 'estimated-stack-usage' := '500'}
METHOD Halt
    _seq.Halt();
END_METHOD

END_FUNCTION_BLOCK

(* ---- FB_MaterialPurgeHMSequence.st ---- *)
FUNCTION_BLOCK PUBLIC FB_MaterialPurgeHMSequence IMPLEMENTS I_TreeNode
VAR
    _seq : FB_SequenceNode;
    // Preparation
    stepCloseNozzle        : FB_CloseValveNode;
    stepClosePCV           : FB_SetControllerNode;

    // Purge cycles (n-1 times)
    stepCyclesRepeat       : FB_RepeatNode;
    stepCycleSeq           : FB_SequenceNode;
    stepDepressurizeHM     : FB_DepressurizeHMSequence;
    stepPressurizeHM       : FB_PressurizeHMSequence;

    // Final cycle
    stepFinalDepressurize  : FB_DepressurizeHMSequence;
    stepFinalPressurize    : FB_PressurizeHMSequence;

    // Internal state
    _bInitialized          : BOOL := FALSE;
    _eSide                 : E_GasSide;
END_VAR

VAR CONSTANT
    DEFAULT_PURGE_CYCLES : INT := 2;
END_VAR

METHOD PUBLIC Init : BOOL
VAR_INPUT
    ipProvider      : I_HardwareProvider;
    eSide           : E_GasSide;
END_VAR
VAR
    ipPCV            : I_Controller;
    ipNozzleIso      : I_Valve;
    ipHMPurge        : I_Valve;
    ipHMVacuumIso    : I_Valve;
    ipHMPressure     : I_Sensor;
END_VAR
    IF _bInitialized THEN
        IF _eSide = eSide THEN
            Init := TRUE;
            RETURN;
        END_IF
        _seq.ClearChildren();
        stepCycleSeq.ClearChildren();
        _bInitialized := FALSE;
    END_IF

    IF ipProvider = 0 THEN
        GVL_ErrorLogger.Logger.LogError('FB_MaterialPurgeHMSequence', E_ErrorId.ERR_GEN_NULL_POINTER, 'Provider is null');
        RETURN;
    END_IF
    _eSide := eSide;

    // Resolve hardware for prep
    ipPCV := ipProvider.GetPressureController(eSide);
    ipNozzleIso := ipProvider.GetNozzleIsoValve(eSide);
    ipHMPurge := ipProvider.GetHMPurgeValve(eSide);
    ipHMVacuumIso := ipProvider.GetHMVacuumIsoValve(eSide);
    ipHMPressure := ipProvider.GetHMPressureSensor(eSide);

    // Validate hardware
    IF ipPCV = 0 OR ipNozzleIso = 0 OR ipHMPurge = 0 OR ipHMVacuumIso = 0 OR ipHMPressure = 0 THEN
        GVL_ErrorLogger.Logger.LogError('FB_MaterialPurgeHMSequence', E_ErrorId.ERR_GEN_NULL_POINTER, 'Hardware reference is null');
        RETURN;
    END_IF

    // Preparation: close boundaries
    stepCloseNozzle.Init(ipNozzleIso, sNodeName := 'CloseNozzle');
    _seq.AddChild(stepCloseNozzle);

    stepClosePCV.Init(ipController := ipPCV, rSetpoint := GVL_SequenceConstants.PCV_CLOSED_SETPOINT, sNodeName := 'ClosePCV');
    _seq.AddChild(stepClosePCV);

    // Purge cycles: depressurize then pressurize (n-1 times)
    stepCycleSeq.ClearChildren();

    stepDepressurizeHM.Init(ipProvider := ipProvider, eSide := eSide);
    stepDepressurizeHM.NodeName := 'DepressurizeHM';
    stepCycleSeq.AddChild(stepDepressurizeHM);

    stepPressurizeHM.Init(ipProvider := ipProvider, eSide := eSide);
    stepPressurizeHM.NodeName := 'PressurizeHM';
    stepCycleSeq.AddChild(stepPressurizeHM);

    stepCyclesRepeat.SetChild(stepCycleSeq);
    stepCyclesRepeat.nNumCycles := DEFAULT_PURGE_CYCLES;
    stepCyclesRepeat.sName := 'HMPurgeCycles';
    _seq.AddChild(stepCyclesRepeat);

    // Final cycle: end at operating pressure
    stepFinalDepressurize.Init(ipProvider := ipProvider, eSide := eSide);
    stepFinalDepressurize.NodeName := 'FinalDepressurizeHM';
    _seq.AddChild(stepFinalDepressurize);

    stepFinalPressurize.Init(ipProvider := ipProvider, eSide := eSide);
    stepFinalPressurize.NodeName := 'FinalPressurizeHM';
    _seq.AddChild(stepFinalPressurize);

    _seq.sName := CONCAT('PurgeHM_', TO_STRING(eSide));
    _bInitialized := TRUE;
    Init := TRUE;
END_METHOD

METHOD PUBLIC SetParams
VAR_INPUT
    nPurgeCycles            : INT;
    rPurgeFlowRate          : LREAL;
    rPurgePressure          : LREAL;
    rFinalPressure          : LREAL;   // Operating pressure for final pressurization
    rEvacuationPressure     : LREAL;
    tPressurizationTimeout  : TIME;
    tEvacuationTimeout      : TIME;
END_VAR
VAR
    nCycleRepeatCount : INT;
END_VAR
    IF NOT _bInitialized THEN RETURN; END_IF

    // Calculate repeat count: nPurgeCycles - 1 (because we have n-1 repeats plus 1 final)
    IF nPurgeCycles > 1 THEN
        nCycleRepeatCount := nPurgeCycles - 1;
    ELSE
        nCycleRepeatCount := 1;
    END_IF

    stepCyclesRepeat.nNumCycles := nCycleRepeatCount;

    stepPressurizeHM.SetParams(
        rTargetCMPressure := 0.0,
        rTargetHMPressure := rPurgePressure,
        rFlowRate := rPurgeFlowRate,
        tCMPressureTimeout := tPressurizationTimeout,
        tHMPressureTimeout := tPressurizationTimeout
    );

    stepDepressurizeHM.SetParams(
        rVacuumThreshold := rEvacuationPressure,
        tTimeout := tEvacuationTimeout
    );

    stepFinalDepressurize.SetParams(
        rVacuumThreshold := rEvacuationPressure,
        tTimeout := tEvacuationTimeout
    );

    // Final pressurization uses operating pressure, not purge pressure
    stepFinalPressurize.SetParams(
        rTargetCMPressure := 0.0,
        rTargetHMPressure := rFinalPressure,
        rFlowRate := rPurgeFlowRate,
        tCMPressureTimeout := tPressurizationTimeout,
        tHMPressureTimeout := tPressurizationTimeout
    );
END_METHOD

PROPERTY PUBLIC NodeName : STRING(50)
    GET
        NodeName := _seq.sName;
    END_GET
    SET
        _seq.sName := NodeName;
    END_SET
END_PROPERTY

METHOD Tick : ST_NodeResult
    IF NOT _bInitialized THEN
        Tick.eStatus := E_NodeStatus.FAILURE;
        Tick.bHasError := TRUE;
        Tick.stError.eErrorId := E_ErrorId.ERR_GEN_INITIALIZATION;
        Tick.stError.sSource := 'FB_MaterialPurgeHMSequence';
        Tick.stError.sMessage := 'Init must be called before Tick';
        Tick.sDescription := Tick.stError.sMessage;
        RETURN;
    END_IF

    Tick := _seq.Tick();
END_METHOD

{attribute 'estimated-stack-usage' := '500'}
METHOD Reset : BOOL
    Reset := _seq.Reset();
END_METHOD

{attribute 'estimated-stack-usage' := '500'}
METHOD Halt
    _seq.Halt();
END_METHOD

END_FUNCTION_BLOCK

(* ---- FB_MaterialPurgeUmbilicalSequence.st ---- *)
FUNCTION_BLOCK PUBLIC FB_MaterialPurgeUmbilicalSequence IMPLEMENTS I_TreeNode
VAR
    _seq : FB_SequenceNode;
    // Phase 1: Preparation
    stepCloseNozzleIso     : FB_CloseValveNode;
    stepClosePCV           : FB_SetControllerNode;

    // Phase 2: Pressurize via purge bypass (CM->HM to prevent backflow)
    stepOpenGasIso         : FB_OpenValveNode;
    stepSetMFC             : FB_SetControllerNode;
    stepOpenCMPurge        : FB_OpenValveNode;
    stepWaitForCMPressure  : FB_WaitForSensorNode;
    stepOpenHMPurge        : FB_OpenValveNode;
    stepWaitForHMPressure  : FB_WaitForSensorNode;

    // Phase 3: Purge to atmosphere
    stepSetPCV             : FB_SetControllerNode;
    stepStabilizationDelay : FB_WaitNode;
    stepOpenNozzleIso      : FB_OpenValveNode;
    stepPurgeDuration      : FB_WaitNode;

    // Phase 4: Cleanup
    stepCleanup            : FB_SequenceNode;
    stepCloseNozzleIsoFinal: FB_CloseValveNode;
    stepClosePCVFinal      : FB_SetControllerNode;
    stepStopMFC            : FB_SetControllerNode;
    stepCloseGasIso        : FB_CloseValveNode;
    stepCloseCMPurge       : FB_CloseValveNode;
    stepCloseHMPurge       : FB_CloseValveNode;

    // Internal state
    _bInitialized          : BOOL := FALSE;
    _bParamsConfigured     : BOOL := FALSE;
    _eSide                 : E_GasSide;
END_VAR

VAR CONSTANT
    DEFAULT_STABILIZATION_DELAY : TIME := T#5S;
    DEFAULT_PURGE_DURATION      : TIME := T#30S;
END_VAR

METHOD PUBLIC Init : BOOL
VAR_INPUT
    ipProvider : I_HardwareProvider;
    eSide      : E_GasSide;
END_VAR
VAR
    ipGasIso      : I_Valve;
    ipMFC         : I_Controller;
    ipCMPurge     : I_Valve;
    ipCMPressure  : I_Sensor;
    ipHMPurge     : I_Valve;
    ipHMPressure  : I_Sensor;
    ipPCV         : I_Controller;
    ipNozzleIso   : I_Valve;
END_VAR
    IF _bInitialized THEN
        IF _eSide = eSide THEN
            Init := TRUE;
            RETURN;
        END_IF
        _seq.ClearChildren();
        stepCleanup.ClearChildren();
        _bInitialized := FALSE;
    END_IF

    IF ipProvider = 0 THEN
        GVL_ErrorLogger.Logger.LogError('FB_MaterialPurgeUmbilicalSequence', E_ErrorId.ERR_GEN_NULL_POINTER, 'Provider is null');
        RETURN;
    END_IF
    _eSide := eSide;

    // Resolve hardware
    ipGasIso := ipProvider.GetGasIsoValve(eSide, 0);
    ipMFC := ipProvider.GetMFCController(eSide);
    ipCMPurge := ipProvider.GetCMPurgeValve(eSide);
    ipCMPressure := ipProvider.GetCMPressureSensor(eSide);
    ipHMPurge := ipProvider.GetHMPurgeValve(eSide);
    ipHMPressure := ipProvider.GetHMPressureSensor(eSide);
    ipPCV := ipProvider.GetPressureController(eSide);
    ipNozzleIso := ipProvider.GetNozzleIsoValve(eSide);

    // Validate hardware
    IF ipGasIso = 0 OR ipMFC = 0 OR ipCMPurge = 0 OR ipCMPressure = 0 OR
       ipHMPurge = 0 OR ipHMPressure = 0 OR ipPCV = 0 OR ipNozzleIso = 0 THEN
        GVL_ErrorLogger.Logger.LogError('FB_MaterialPurgeUmbilicalSequence', E_ErrorId.ERR_GEN_NULL_POINTER, 'Hardware reference is null');
        RETURN;
    END_IF

    // Phase 1: Preparation
    stepCloseNozzleIso.Init(ipNozzleIso, sNodeName := 'CloseNozzleIso');
    _seq.AddChild(stepCloseNozzleIso);

    stepClosePCV.Init(ipController := ipPCV, rSetpoint := GVL_SequenceConstants.PCV_CLOSED_SETPOINT, sNodeName := 'ClosePCV');
    _seq.AddChild(stepClosePCV);

    // Phase 2: Pressurize via purge bypass (CM->HM to prevent backflow)
    stepOpenGasIso.Init(ipGasIso, sNodeName := 'OpenGasIso');
    _seq.AddChild(stepOpenGasIso);

    stepSetMFC.Init(ipController := ipMFC, rSetpoint := 0.0, sNodeName := 'SetPurgeMFC');
    _seq.AddChild(stepSetMFC);

    stepOpenCMPurge.Init(ipCMPurge, sNodeName := 'OpenCMPurge');
    _seq.AddChild(stepOpenCMPurge);

    // Wait for CM pressure before opening HM to prevent backflow
    stepWaitForCMPressure.Init(ipSensor := ipCMPressure, rTarget := 0.0, eMode := E_CompareMode.GREATER_THAN, sNodeName := 'WaitForCMPressure');
    _seq.AddChild(stepWaitForCMPressure);

    stepOpenHMPurge.Init(ipHMPurge, sNodeName := 'OpenHMPurge');
    _seq.AddChild(stepOpenHMPurge);

    stepWaitForHMPressure.Init(ipSensor := ipHMPressure, rTarget := 0.0, eMode := E_CompareMode.GREATER_THAN, sNodeName := 'WaitForHMPressure');
    _seq.AddChild(stepWaitForHMPressure);

    // Phase 3: Purge to atmosphere
    stepSetPCV.Init(ipController := ipPCV, rSetpoint := 0.0, sNodeName := 'SetPCVSetpoint');
    _seq.AddChild(stepSetPCV);

    stepStabilizationDelay.Init(tWaitTime := DEFAULT_STABILIZATION_DELAY, sNodeName := 'StabilizationDelay');
    _seq.AddChild(stepStabilizationDelay);

    stepOpenNozzleIso.Init(ipNozzleIso, sNodeName := 'OpenNozzleIso');
    _seq.AddChild(stepOpenNozzleIso);

    stepPurgeDuration.Init(tWaitTime := DEFAULT_PURGE_DURATION, sNodeName := 'PurgeDuration');
    _seq.AddChild(stepPurgeDuration);

    // Phase 4: Cleanup
    stepCleanup.ClearChildren();

    stepCloseNozzleIsoFinal.Init(ipNozzleIso, sNodeName := 'CloseNozzleIsoFinal');
    stepCleanup.AddChild(stepCloseNozzleIsoFinal);

    stepClosePCVFinal.Init(ipController := ipPCV, rSetpoint := GVL_SequenceConstants.PCV_CLOSED_SETPOINT, sNodeName := 'ClosePCVFinal');
    stepCleanup.AddChild(stepClosePCVFinal);

    stepStopMFC.Init(ipController := ipMFC, rSetpoint := 0.0, sNodeName := 'StopMFC');
    stepCleanup.AddChild(stepStopMFC);

    stepCloseGasIso.Init(ipGasIso, sNodeName := 'CloseGasIso');
    stepCleanup.AddChild(stepCloseGasIso);

    stepCloseCMPurge.Init(ipCMPurge, sNodeName := 'CloseCMPurge');
    stepCleanup.AddChild(stepCloseCMPurge);

    stepCloseHMPurge.Init(ipHMPurge, sNodeName := 'CloseHMPurge');
    stepCleanup.AddChild(stepCloseHMPurge);

    stepCleanup.sName := 'Cleanup';
    _seq.AddChild(stepCleanup);

    _seq.sName := CONCAT('UmbilicalPurge_', TO_STRING(eSide));
    _bParamsConfigured := FALSE;
    _bInitialized := TRUE;
    Init := TRUE;
END_METHOD

METHOD PUBLIC SetParams
VAR_INPUT
    rPurgeFlowRate      : LREAL;
    rCMPressureTarget   : LREAL;
    rHMPressureTarget   : LREAL;
    rPCVSetpoint        : LREAL;
    tCMPressureTimeout  : TIME;
    tHMPressureTimeout  : TIME;
    tStabilizationDelay : TIME;
    tPurgeDuration      : TIME;
END_VAR
    IF NOT _bInitialized THEN RETURN; END_IF

    stepSetMFC.Setpoint := rPurgeFlowRate;

    stepWaitForCMPressure.Target := rCMPressureTarget;
    stepWaitForCMPressure.Timeout := tCMPressureTimeout;

    stepWaitForHMPressure.Target := rHMPressureTarget;
    stepWaitForHMPressure.Timeout := tHMPressureTimeout;

    stepSetPCV.Setpoint := rPCVSetpoint;

    stepStabilizationDelay.WaitTime := tStabilizationDelay;
    stepPurgeDuration.WaitTime := tPurgeDuration;
    _bParamsConfigured := TRUE;
END_METHOD

PROPERTY PUBLIC NodeName : STRING(50)
    GET
        NodeName := _seq.sName;
    END_GET
    SET
        _seq.sName := NodeName;
    END_SET
END_PROPERTY

METHOD Tick : ST_NodeResult
    IF NOT _bInitialized THEN
        Tick.eStatus := E_NodeStatus.FAILURE;
        Tick.bHasError := TRUE;
        Tick.stError.eErrorId := E_ErrorId.ERR_GEN_INITIALIZATION;
        Tick.stError.sSource := 'FB_MaterialPurgeUmbilicalSequence';
        Tick.stError.sMessage := 'Init must be called before Tick';
        Tick.sDescription := Tick.stError.sMessage;
        RETURN;
    END_IF

    IF NOT _bParamsConfigured THEN
        Tick.eStatus := E_NodeStatus.FAILURE;
        Tick.bHasError := TRUE;
        Tick.stError.eErrorId := E_ErrorId.ERR_GEN_NOT_CONFIGURED;
        Tick.stError.sSource := 'FB_MaterialPurgeUmbilicalSequence';
        Tick.stError.sMessage := 'SetParams must be called before Tick';
        Tick.sDescription := Tick.stError.sMessage;
        RETURN;
    END_IF

    Tick := _seq.Tick();
END_METHOD

{attribute 'estimated-stack-usage' := '500'}
METHOD Reset : BOOL
    Reset := _seq.Reset();
END_METHOD

{attribute 'estimated-stack-usage' := '500'}
METHOD Halt
    _seq.Halt();
END_METHOD

END_FUNCTION_BLOCK

(* ---- FB_PrepareExhaustSequence.st ---- *)
FUNCTION_BLOCK PUBLIC FB_PrepareExhaustSequence IMPLEMENTS I_TreeNode
VAR
    _seq : FB_SequenceNode;
    // Steps
    stepTurnOnPump        : FB_SetDigitalOutputNode;
    stepOpenExhaustVacIso : FB_OpenValveNode;
    stepSetPCVInitial     : FB_SetControllerNode;

    // Internal state
    _bInitialized         : BOOL := FALSE;
    _eSide                : E_GasSide;
END_VAR

METHOD PUBLIC Init : BOOL
VAR_INPUT
    ipProvider      : I_HardwareProvider;
    eSide           : E_GasSide;
END_VAR
    IF _bInitialized THEN
        IF _eSide = eSide THEN
            Init := TRUE;
            RETURN;
        END_IF
        _bInitialized := FALSE;
    END_IF

    IF ipProvider = 0 THEN
        GVL_ErrorLogger.Logger.LogError('FB_PrepareExhaustSequence', E_ErrorId.ERR_GEN_NULL_POINTER, 'Provider is null');
        RETURN;
    END_IF
    _eSide := eSide;

    _seq.ClearChildren();

    stepTurnOnPump.Init(ipDO := ipProvider.GetExhaustPump(), bState := TRUE, sNodeName := 'TurnOnExhaustPump');
    _seq.AddChild(stepTurnOnPump);

    stepOpenExhaustVacIso.Init(ipProvider.GetExhaustVacuumIsoValve(), sNodeName := 'OpenExhaustVacIso');
    _seq.AddChild(stepOpenExhaustVacIso);

    // Set PCV to fully open for unrestricted exhaust flow
    stepSetPCVInitial.Init(ipController := ipProvider.GetPressureController(eSide), rSetpoint := GVL_SequenceConstants.PCV_OPEN_SETPOINT, sNodeName := 'SetPCVOpen');
    _seq.AddChild(stepSetPCVInitial);

    _seq.sName := 'PrepareExhaust';
    _bInitialized := TRUE;
    Init := TRUE;
END_METHOD

PROPERTY PUBLIC NodeName : STRING(50)
    GET
        NodeName := _seq.sName;
    END_GET
    SET
        _seq.sName := NodeName;
    END_SET
END_PROPERTY

METHOD Tick : ST_NodeResult
    IF NOT _bInitialized THEN
        Tick.eStatus := E_NodeStatus.FAILURE;
        Tick.bHasError := TRUE;
        Tick.stError.eErrorId := E_ErrorId.ERR_GEN_INITIALIZATION;
        Tick.stError.sSource := 'FB_PrepareExhaustSequence';
        Tick.stError.sMessage := 'Init must be called before Tick';
        Tick.sDescription := Tick.stError.sMessage;
        RETURN;
    END_IF

    Tick := _seq.Tick();
END_METHOD

{attribute 'estimated-stack-usage' := '500'}
METHOD Reset : BOOL
    Reset := _seq.Reset();
END_METHOD

{attribute 'estimated-stack-usage' := '500'}
METHOD Halt
    _seq.Halt();
END_METHOD

END_FUNCTION_BLOCK

(* ---- FB_PressurizeCMSequence.st ---- *)
FUNCTION_BLOCK PUBLIC FB_PressurizeCMSequence IMPLEMENTS I_TreeNode
VAR
    _seq : FB_SequenceNode;
    // Steps
    stepCloseNozzle        : FB_CloseValveNode;    // Isolate from process
    stepClosePCV           : FB_SetControllerNode; // Isolate from exhaust
    stepOpenGasIso         : FB_OpenValveNode;     // Supply
    stepSetMFC             : FB_SetControllerNode; // Flow
    stepOpenCMPurge        : FB_OpenValveNode;     // Path into CM
    stepWaitForPressure    : FB_WaitForSensorNode;
    stepCloseCMPurge       : FB_CloseValveNode;    // Isolate after fill
    stepCloseGasIso        : FB_CloseValveNode;
    stepStopMFC            : FB_SetControllerNode;

    // Internal state
    _bInitialized             : BOOL := FALSE;
    _bParamsConfigured        : BOOL := FALSE;
    _eSide                    : E_GasSide;
END_VAR

METHOD PUBLIC Init : BOOL
VAR_INPUT
    ipProvider      : I_HardwareProvider;
    eSide           : E_GasSide;
END_VAR
VAR
    ipGasIso         : I_Valve;
    ipCMPurge        : I_Valve;
    ipNozzleIso      : I_Valve;
    ipCMPressure     : I_Sensor;
    ipMFC            : I_Controller;
END_VAR
    IF _bInitialized THEN
        IF _eSide = eSide THEN
            Init := TRUE;
            RETURN;
        END_IF
        _seq.ClearChildren();
        _bInitialized := FALSE;
    END_IF

    IF ipProvider = 0 THEN
        GVL_ErrorLogger.Logger.LogError('FB_PressurizeCMSequence', E_ErrorId.ERR_GEN_NULL_POINTER, 'Provider is null');
        RETURN;
    END_IF
    _eSide := eSide;

    ipMFC := ipProvider.GetMFCController(eSide);
    ipGasIso := ipProvider.GetGasIsoValve(eSide, 0);
    ipCMPurge := ipProvider.GetCMPurgeValve(eSide);
    ipNozzleIso := ipProvider.GetNozzleIsoValve(eSide);
    ipCMPressure := ipProvider.GetCMPressureSensor(eSide);

    IF ipMFC = 0 OR ipGasIso = 0 OR ipCMPurge = 0 OR ipNozzleIso = 0 OR ipCMPressure = 0 THEN
        GVL_ErrorLogger.Logger.LogError('FB_PressurizeCMSequence', E_ErrorId.ERR_GEN_NULL_POINTER, 'Hardware reference is null');
        RETURN;
    END_IF

    // Secure boundaries before pressurizing
    stepCloseNozzle.Init(ipNozzleIso, sNodeName := 'CloseNozzle');
    _seq.AddChild(stepCloseNozzle);

    stepClosePCV.Init(ipController := ipProvider.GetPressureController(eSide), rSetpoint := GVL_SequenceConstants.PCV_CLOSED_SETPOINT, sNodeName := 'ClosePCV');
    _seq.AddChild(stepClosePCV);

    // Open supply and set flow
    stepOpenGasIso.Init(ipGasIso, sNodeName := 'OpenGasIso');
    _seq.AddChild(stepOpenGasIso);

    stepSetMFC.Init(ipController := ipMFC, rSetpoint := 0.0, sNodeName := 'SetMFC');
    _seq.AddChild(stepSetMFC);

    // Pressurize CM
    stepOpenCMPurge.Init(ipCMPurge, sNodeName := 'OpenCMPurge');
    _seq.AddChild(stepOpenCMPurge);

    stepWaitForPressure.Init(ipSensor := ipCMPressure, rTarget := 0.0, eMode := E_CompareMode.GREATER_THAN, sNodeName := 'WaitCMPressure');
    _seq.AddChild(stepWaitForPressure);

    // Cleanup
    stepCloseCMPurge.Init(ipCMPurge, sNodeName := 'IsolateCM');
    _seq.AddChild(stepCloseCMPurge);

    stepCloseGasIso.Init(ipGasIso, sNodeName := 'CloseGasIso');
    _seq.AddChild(stepCloseGasIso);

    stepStopMFC.Init(ipController := ipMFC, rSetpoint := 0.0, sNodeName := 'StopMFC');
    _seq.AddChild(stepStopMFC);

    _seq.sName := CONCAT('PressurizeCM_', TO_STRING(eSide));
    _bParamsConfigured := FALSE;
    _bInitialized := TRUE;
    Init := TRUE;
END_METHOD

METHOD PUBLIC SetParams
VAR_INPUT
    rTargetPressure  : LREAL;
    rFlowRate        : LREAL;
    tTimeout         : TIME;
END_VAR
    IF NOT _bInitialized THEN RETURN; END_IF

    stepSetMFC.Setpoint := rFlowRate;
    stepWaitForPressure.Target := rTargetPressure;
    stepWaitForPressure.Timeout := tTimeout;
    _bParamsConfigured := TRUE;
END_METHOD

PROPERTY PUBLIC NodeName : STRING(50)
    GET
        NodeName := _seq.sName;
    END_GET
    SET
        _seq.sName := NodeName;
    END_SET
END_PROPERTY

METHOD Tick : ST_NodeResult
    IF NOT _bInitialized THEN
        Tick.eStatus := E_NodeStatus.FAILURE;
        Tick.bHasError := TRUE;
        Tick.stError.eErrorId := E_ErrorId.ERR_GEN_INITIALIZATION;
        Tick.stError.sSource := 'FB_PressurizeCMSequence';
        Tick.stError.sMessage := 'Init must be called before Tick';
        Tick.sDescription := Tick.stError.sMessage;
        RETURN;
    END_IF

    IF NOT _bParamsConfigured THEN
        Tick.eStatus := E_NodeStatus.FAILURE;
        Tick.bHasError := TRUE;
        Tick.stError.eErrorId := E_ErrorId.ERR_GEN_NOT_CONFIGURED;
        Tick.stError.sSource := 'FB_PressurizeCMSequence';
        Tick.stError.sMessage := 'SetParams must be called before Tick';
        Tick.sDescription := Tick.stError.sMessage;
        RETURN;
    END_IF

    Tick := _seq.Tick();
END_METHOD

{attribute 'estimated-stack-usage' := '500'}
METHOD Reset : BOOL
    Reset := _seq.Reset();
END_METHOD

{attribute 'estimated-stack-usage' := '500'}
METHOD Halt
    _seq.Halt();
END_METHOD

END_FUNCTION_BLOCK

(* ---- FB_PressurizeHMSequence.st ---- *)
FUNCTION_BLOCK PUBLIC FB_PressurizeHMSequence IMPLEMENTS I_TreeNode
VAR
    _seq : FB_SequenceNode;
    // Safety and supply
    stepCloseNozzle     : FB_CloseValveNode;
    stepClosePCV        : FB_SetControllerNode;
    stepOpenGasIso      : FB_OpenValveNode;
    stepSetMFCBuildupFlow : FB_SetControllerNode;

    // Initial gas pressure buildup
    stepWaitGasPressure : FB_WaitForSensorNode;

    // CM pressure buildup
    stepOpenCMPurge     : FB_OpenValveNode;
    stepWaitCMPressure  : FB_WaitForSensorNode;

    // HM pressurization
    stepOpenHMPurge     : FB_OpenValveNode;
    stepWaitHMPressure  : FB_WaitForSensorNode;

    // Cleanup (reverse order)
    stepCloseHMPurge    : FB_CloseValveNode;
    stepCloseCMPurge    : FB_CloseValveNode;
    stepZeroMFC         : FB_SetControllerNode;
    stepCloseGasIso     : FB_CloseValveNode;

    // Internal state
    _bInitialized          : BOOL := FALSE;
    _bParamsConfigured     : BOOL := FALSE;
    _eSide                 : E_GasSide;
END_VAR

METHOD PUBLIC Init : BOOL
VAR_INPUT
    ipProvider          : I_HardwareProvider;
    eSide               : E_GasSide;
    tCMPressureTimeout  : TIME  := T#10M;
    tHMPressureTimeout  : TIME  := T#10M;
END_VAR
VAR
    ipGasIso            : I_Valve;
    ipCMPurge           : I_Valve;
    ipHMPurge           : I_Valve;
    ipNozzleIso         : I_Valve;
    ipMFC               : I_Controller;
    ipPCV               : I_Controller;
    ipCMPressureSensor  : I_Sensor;
    ipHMPressureSensor  : I_Sensor;
END_VAR
    IF _bInitialized THEN
        IF _eSide = eSide THEN
            Init := TRUE;
            RETURN;
        END_IF
        _seq.ClearChildren();
        _bInitialized := FALSE;
    END_IF

    IF ipProvider = 0 THEN
        GVL_ErrorLogger.Logger.LogError('FB_PressurizeHMSequence', E_ErrorId.ERR_GEN_NULL_POINTER, 'Provider is null');
        RETURN;
    END_IF
    _eSide := eSide;

    // Resolve hardware references
    ipMFC := ipProvider.GetMFCController(eSide);
    ipGasIso := ipProvider.GetGasIsoValve(eSide, 0);
    ipCMPurge := ipProvider.GetCMPurgeValve(eSide);
    ipHMPurge := ipProvider.GetHMPurgeValve(eSide);
    ipNozzleIso := ipProvider.GetNozzleIsoValve(eSide);
    ipPCV := ipProvider.GetPressureController(eSide);
    ipCMPressureSensor := ipProvider.GetCMPressureSensor(eSide);
    ipHMPressureSensor := ipProvider.GetHMPressureSensor(eSide);

    IF ipMFC = 0 OR ipGasIso = 0 OR ipCMPurge = 0 OR ipHMPurge = 0 OR ipNozzleIso = 0 OR
       ipPCV = 0 OR ipCMPressureSensor = 0 OR ipHMPressureSensor = 0 THEN
        GVL_ErrorLogger.Logger.LogError('FB_PressurizeHMSequence', E_ErrorId.ERR_GEN_NULL_POINTER, 'Hardware reference is null');
        RETURN;
    END_IF

    // Safety: close nozzle and PCV before pressurizing
    stepCloseNozzle.Init(ipNozzleIso, sNodeName := 'CloseNozzle');
    _seq.AddChild(stepCloseNozzle);

    stepClosePCV.Init(ipController := ipPCV, rSetpoint := GVL_SequenceConstants.PCV_CLOSED_SETPOINT, sNodeName := 'ClosePCV');
    _seq.AddChild(stepClosePCV);

    // Open supply
    stepOpenGasIso.Init(ipGasIso, sNodeName := 'OpenGasIso');
    _seq.AddChild(stepOpenGasIso);

    stepSetMFCBuildupFlow.Init(ipController := ipMFC, rSetpoint := 0.0, sNodeName := 'SetMFCBuildup');
    _seq.AddChild(stepSetMFCBuildupFlow);

    // Wait for initial gas pressure before opening CM Purge
    stepWaitGasPressure.Init(ipSensor := ipCMPressureSensor, rTarget := 0.0, eMode := E_CompareMode.GREATER_THAN, tTimeout := tCMPressureTimeout, sNodeName := 'WaitGasPressure');
    _seq.AddChild(stepWaitGasPressure);

    // Build CM pressure
    stepOpenCMPurge.Init(ipCMPurge, sNodeName := 'OpenCMPurge');
    _seq.AddChild(stepOpenCMPurge);

    stepWaitCMPressure.Init(ipSensor := ipCMPressureSensor, rTarget := 0.0, eMode := E_CompareMode.GREATER_THAN, tTimeout := tCMPressureTimeout, sNodeName := 'WaitCMPressure');
    _seq.AddChild(stepWaitCMPressure);

    // Pressurize HM
    stepOpenHMPurge.Init(ipHMPurge, sNodeName := 'OpenHMPurge');
    _seq.AddChild(stepOpenHMPurge);

    stepWaitHMPressure.Init(ipSensor := ipHMPressureSensor, rTarget := 0.0, eMode := E_CompareMode.GREATER_THAN, tTimeout := tHMPressureTimeout, sNodeName := 'WaitHMPressure');
    _seq.AddChild(stepWaitHMPressure);

    // Cleanup in reverse order
    stepCloseHMPurge.Init(ipHMPurge, sNodeName := 'IsolateHM');
    _seq.AddChild(stepCloseHMPurge);

    stepCloseCMPurge.Init(ipCMPurge, sNodeName := 'CloseCMPurge');
    _seq.AddChild(stepCloseCMPurge);

    stepZeroMFC.Init(ipController := ipMFC, rSetpoint := 0.0, sNodeName := 'ZeroMFC');
    _seq.AddChild(stepZeroMFC);

    stepCloseGasIso.Init(ipGasIso, sNodeName := 'CloseGasIso');
    _seq.AddChild(stepCloseGasIso);

    _seq.sName := CONCAT('PressurizeHM_', TO_STRING(eSide));
    _bParamsConfigured := FALSE;
    _bInitialized := TRUE;
    Init := TRUE;
END_METHOD

METHOD PUBLIC SetParams
VAR_INPUT
    rTargetCMPressure   : LREAL;   // Target CM pressure
    rTargetHMPressure   : LREAL;   // Target HM pressure (full pressurize)
    rFlowRate           : LREAL;   // MFC buildup flow rate (sccm)
    tCMPressureTimeout  : TIME;    // Timeout for CM pressure buildup
    tHMPressureTimeout  : TIME;
END_VAR
    IF NOT _bInitialized THEN RETURN; END_IF

    stepSetMFCBuildupFlow.Setpoint := rFlowRate;

    stepWaitGasPressure.Target := rTargetCMPressure;
    stepWaitGasPressure.Timeout := tCMPressureTimeout;

    stepWaitCMPressure.Target := rTargetCMPressure;
    stepWaitCMPressure.Timeout := tCMPressureTimeout;

    stepWaitHMPressure.Target := rTargetHMPressure;
    stepWaitHMPressure.Timeout := tHMPressureTimeout;
    _bParamsConfigured := TRUE;
END_METHOD

PROPERTY PUBLIC NodeName : STRING(50)
    GET
        NodeName := _seq.sName;
    END_GET
    SET
        _seq.sName := NodeName;
    END_SET
END_PROPERTY

METHOD Tick : ST_NodeResult
    IF NOT _bInitialized THEN
        Tick.eStatus := E_NodeStatus.FAILURE;
        Tick.bHasError := TRUE;
        Tick.stError.eErrorId := E_ErrorId.ERR_GEN_INITIALIZATION;
        Tick.stError.sSource := 'FB_PressurizeHMSequence';
        Tick.stError.sMessage := 'Init must be called before Tick';
        Tick.sDescription := Tick.stError.sMessage;
        RETURN;
    END_IF

    IF NOT _bParamsConfigured THEN
        Tick.eStatus := E_NodeStatus.FAILURE;
        Tick.bHasError := TRUE;
        Tick.stError.eErrorId := E_ErrorId.ERR_GEN_NOT_CONFIGURED;
        Tick.stError.sSource := 'FB_PressurizeHMSequence';
        Tick.stError.sMessage := 'SetParams must be called before Tick';
        Tick.sDescription := Tick.stError.sMessage;
        RETURN;
    END_IF

    Tick := _seq.Tick();
END_METHOD

{attribute 'estimated-stack-usage' := '500'}
METHOD Reset : BOOL
    Reset := _seq.Reset();
END_METHOD

{attribute 'estimated-stack-usage' := '500'}
METHOD Halt
    _seq.Halt();
END_METHOD

END_FUNCTION_BLOCK
